PROGRAM MAIN
VAR
	bInit: BOOL := TRUE;
	fbSocketCloseAll: FB_SocketCloseAll; 
	bSocketCloseError: BOOL;
	nSocketCloseError: UDINT;	
	nServer1Port				: UDINT 				:= 5050;
	sServer1Host				: T_IPv4Addr 			:= '';		
		
	fbTcpEchoServer1				: FB_TCPServer;
		sServerReceivedData			: STRING(255);
		bStartServer1Communication	: BOOL 					:= TRUE;
		bServer1Connected			: BOOL;
		sServerData					: STRING(255);
		bServer1Busy				: BOOL;
		bServer1Error				: BOOL;
		nServer1ErrorID				: UDINT;
	
	bAutogenerateData				: BOOL 					:= TRUE;
	fbTimer1						: TON;
	nCnt							: UDINT;
END_VAR

IF bInit THEN 				// Init Step to close all sockets after login PLC with  downlaod
	fbSocketCloseAll(
		sSrvNetId:= '', 
		bExecute:= TRUE, 
		tTimeout:= T#3S, 
		bBusy=> , 
		bError=> bSocketCloseError, 
		nErrId=> nSocketCloseError);
	IF NOT (fbSocketCloseAll.bBusy OR fbSocketCloseAll.bError) THEN
		bInit := FALSE;
		fbSocketCloseAll(bExecute:= FALSE);
	END_IF
ELSE
		
	fbTcpEchoServer1(
		sLocalHost:= '192.168.17.110', 											// Server IP Adress
		nLocalPort:= nServer1Port, 									// Server port
		bStartCommunication:= bStartServer1Communication, 			// Allow Client-connection or close connection
		bConnected => bServer1Connected,							// Client connection is valid
		sSendData => sServerData,
		bBusy=> bServer1Busy, 
		bError=> bServer1Error, 
		nErrorID=> nServer1ErrorID);
END_IF

END_PROGRAM

(* stored: Version 1.1.0.1, ProductVersion 3.1.4024.12
   POU MAIN: Id {572507de-a44a-4a7e-b7eb-52f2373576ea}, SpecialFunc None *)
